Fanuc KAREL source: kb00170.KL

-- PROVISIONAL review KL for V940-1; original PC SHA256 76d5ebbdc6c07201555b26bf97c887edd364f700d87f7530b0fc14bad1bee799
-- Incomplete behavior may be omitted. Consult companion uncertainty JSON. Do not deploy.
PROGRAM KB00170
%NOLOCKGROUP
BEGIN
  -- V9_ZERO_TABLE_METADATA_HINT layout=0002_ascii; no indexed target words; source/name/runtime held
  -- UNRESOLVED_PC offsets 5-12; opcodes 9D,23
  -- UNRESOLVED_PC offsets 17-24; opcodes 9D,23
  -- UNRESOLVED_PC offsets 29-36; opcodes 9D,23
  -- UNRESOLVED_PC offsets 41-48; opcodes 9D,23
  -- UNRESOLVED_PC offsets 53-60; opcodes 9D,23
  -- UNRESOLVED_PC offsets 65-72; opcodes 9D,23
  -- UNRESOLVED_PC offsets 77-84; opcodes 9D,23
  -- UNRESOLVED_PC offsets 89-96; opcodes 9D,23
  -- UNRESOLVED_PC offsets 101-153; opcodes 27,22,22,22,22,22,22,22,22,31
  -- UNRESOLVED_PC offsets 158-162; opcodes 7F
END KB00170
